INTERFACE ITF_1_Tool

METHOD Grip : BOOL
VAR_INPUT
END_VAR
END_METHOD

METHOD Release : BOOL
VAR_INPUT
END_VAR
END_METHOD

END_INTERFACE

(* stored: Version 1.1.0.1, ProductVersion 3.1.4026.18
   Itf ITF_1_Tool: Id {401e2f37-a48a-4601-b049-191cb683eebc}
   Method Grip: Id {8d9f4c5f-6eec-4f7a-b2a0-780c13b9b5ce}
   Method Release: Id {202fb732-cc5b-491e-89c1-ded2a24699ec} *)
